# EPICS IOC start-up script: iocsh/Pelco_CM6700.iocsh
# ### Pelco_CM6700.iocsh ###

#- ###################################################
#- PREFIX         - IOC Prefix
#- INSTANCE       - Instance Prefix
#- PORT           - Serial port name
#- IP             - Location of IP module
#- SUB            - Optional: Names substitution file (Pelco_CM6700_names.db)
#-                            Macros P and R will be set automatically.
#-                  Default: $(IP)/iocsh/Pelco_CM6700_default.substitutions
#- ###################################################

iocshLoad("$(IP)/iocsh/setSerialParams.iocsh", "BAUD=9600, BITS=8, STOP=1, PARITY=odd")

asynOctetSetInputEos( "$(PORT)", -1, "")
asynOctetSetOutputEos("$(PORT)", -1, "")

dbLoadRecords("$(IP)/ipApp/Db/Pelco_CM6700.db", "P=$(PREFIX),R=$(INSTANCE),PORT=$(PORT)")
dbLoadTemplate("$(SUB=$(IP)/iocsh/Pelco_CM6700_default.substitutions)", "P=$(PREFIX),R=$(INSTANCE)")
